FUNCTION_BLOCK MoverSequence
VAR_INPUT
	ThisMover : IMover;
END_VAR
VAR_OUTPUT
END_VAR
VAR
	State :(
        Init,                                               
        Available,                                  
        ForwardMove,
		ForwardStationary,
		ForwardDone,
		ForwardFailed,
		ForwardAborted,
		BackwardMove,
		BackwardStationary,
		BackwardDone,
		BackwardFailed,
		BackwardAborted);  
	
END_VAR

CASE State OF
	State.Init:
	State.Available:
END_CASE

METHOD ClearState : BOOL
VAR_INPUT
END_VAR
ClearCommand := TRUE;
END_METHOD

METHOD SetGroupStop : BOOL
VAR_INPUT
END_VAR
IF _MoverState = XtsMoverStates.ForwardMove OR
		_MoverState = XtsMoverStates.ForwardStationary THEN
	_MoverState := XtsMoverStates.ForwardAborted;
	axesMoveTo.Abort();	
END_IF
IF _MoverState = XtsMoverStates.ReverseMove OR
		_MoverState = XtsMoverStates.ReverseStationary THEN
	_MoverState := XtsMoverStates.ReverseAborted;
	axesMoveTo.Abort();	
END_IF
END_METHOD

METHOD SetStatus : BOOL
VAR_INPUT
END_VAR
IF _MoverState = XtsMoverStates.ForwardMove OR _MoverState = XtsMoverStates.ForwardStationary THEN
	IF _axis.Status.NotMoving THEN
		IF axesMoveTo.Done AND isAtPosition(position := _targetPos) THEN
			_MoverState := XtsMoverStates.ForwardDone;
		ELSE
			_MoverState := XtsMoverStates.ForwardStationary;
		END_IF
	ELSE
		_MoverState := XtsMoverStates.ForwardMove;
	END_IF
END_IF

IF _MoverState = XtsMoverStates.ReverseMove OR _MoverState = XtsMoverStates.ReverseStationary THEN
	IF _axis.Status.NotMoving THEN
		IF axesMoveTo.Done AND isAtPosition(position := _targetPos) THEN
			_MoverState := XtsMoverStates.ReverseDone;
		ELSE
			_MoverState := XtsMoverStates.ReverseStationary;
		END_IF
	ELSE
		_MoverState := XtsMoverStates.ReverseMove;
	END_IF
END_IF


//IF ClearCommand THEN
//	IF _MoverState = XtsMoverStates.ForwardAborted OR
//			_MoverState = XtsMoverStates.ForwardDone OR
//			_MoverState = XtsMoverStates.ReverseAborted OR
//			_MoverState = XtsMoverStates.ForwardFailed OR
//			_MoverState = XtsMoverStates.ReverseFailed OR
//			_MoverState = XtsMoverStates.ReverseDone THEN
//		IF isEnabled() THEN
//			_MoverState := XtsMoverStates.Available;
//		ELSE
//			_MoverState := XtsMoverStates.Idle;
//		END_IF
//	END_IF
	
//	IF _MoverState <> XtsMoverStates.ForwardMove AND	
//			_MoverState <> XtsMoverStates.ForwardStationary AND
//			_MoverState <> XtsMoverStates.ReverseMove AND
//			_MoverState <> XtsMoverStates.ReverseStationary AND 
//			_MoverState <> XtsMoverStates.Idle AND
//			_MoverState <> XtsMoverStates.MoverError THEN
//		_MoverState := XtsMoverStates.Available;
				
//	END_IF
//END_IF

ErrorTrigger(CLK := _axis.Status.Error);
IF ErrorTrigger.Q THEN
	IF _MoverState = XtsMoverStates.ForwardMove OR 
		_MoverState = XtsMoverStates.ForwardStationary THEN
		_MoverState := XtsMoverStates.ForwardFailed;
		axesMoveTo.Abort();
	ELSIF _MoverState = XtsMoverStates.ReverseMove OR
			_MoverState = XtsMoverStates.ReverseStationary THEN
		_MoverState := XtsMoverStates.ReverseFailed;
		axesMoveTo.Abort();
	ELSE
		_MoverState := XtsMoverStates.MoverError;
	END_IF
END_IF

IF _MoverState = XtsMoverStates.MoverError AND NOT _axis.Status.Error THEN
	IF axesEnable.Enable THEN
		IF isEnabled() THEN
			_MoverState := XtsMoverStates.Available;
		END_IF
	ELSE
		_MoverState := XtsMoverStates.Idle;
	END_IF
END_IF
END_METHOD

END_FUNCTION_BLOCK

(* stored: Version 1.1.0.1, ProductVersion 3.1.4024.6
   POU MoverSequence: Id {5b1293cd-307b-4dc9-8f5e-57c564c1904c}, SpecialFunc None
   Method ClearState: Id {a836235b-88fd-4a29-b023-93bff8c050ce}
   Method SetGroupStop: Id {5db54925-4bf7-473d-8e67-6621495b1a92}
   Method SetStatus: Id {3c4ecb94-31de-4ff8-b16b-49e7c8b54463} *)
